// TIA Portal project "TAKT" (V15)

(* hardware
DEVICE "S7-1200 station_1"  S7-1200 Station
   slot 0: "Rack_0"  S7-1200 Rack  Rack  V1.0
   slot 1: "PLC_1"  CPU 1212C DC/DC/DC  6ES7 212-1AE40-0XB0  V4.2
*)

// ===== PLC "PLC_1"  CPU 1212C DC/DC/DC =====

VAR_GLOBAL   // PLC tag table "Default tag table"
   "PULSE1" AT %M0.0 : Bool;
   "PULSE_2" AT %M0.1 : Bool;
   "PULSE_4" AT %M0.2 : Bool;
   "PULSE3" AT %M0.3 : Bool;
END_VAR

TYPE "STOP_TIME"
   STRUCT
      BOTAO_ID : Int;
      DATE_INICIO : DTL;
      DATE_FIM : DTL;
   END_STRUCT;
END_TYPE

DATA_BLOCK "DIA_DA_SEMANA_DB"   // DB2
{ S7_Optimized_Access := 'TRUE' }
VERSION : 0.1
// stored: InstanceOfName DIA_DA_SEMANA
"DIA_DA_SEMANA"
BEGIN
END_DATA_BLOCK

DATA_BLOCK "Takt_Variavel_DB"   // DB4
{ S7_Optimized_Access := 'TRUE' }
VERSION : 0.1
// stored: InstanceOfName Takt_Variavel
"Takt_Variavel"
BEGIN
END_DATA_BLOCK

DATA_BLOCK "BANCO_DADOS_PARADAS"   // DB5
{ S7_Optimized_Access := 'TRUE' }
VERSION : 0.1
   VAR
      STOP_TIME : Array[0..1000] of "STOP_TIME";
   END_VAR
BEGIN
END_DATA_BLOCK

DATA_BLOCK "RELATORIO_DB"   // DB6
{ S7_Optimized_Access := 'TRUE' }
VERSION : 0.1
// stored: InstanceOfName RELATORIO
"RELATORIO"
BEGIN
END_DATA_BLOCK

DATA_BLOCK "TONR_DB"   // DB8
{ S7_Optimized_Access := 'TRUE' }
VERSION : 0.1
// stored: InstanceOfName TONR
"TONR"
BEGIN
END_DATA_BLOCK

// folder: System blocks/Program resources

DATA_BLOCK "Counter_DIA"   // DB1
{ S7_Optimized_Access := 'TRUE' }
AUTHOR : Simatic
FAMILY : IEC
NAME : CNTR
VERSION : 1.0
// stored: InstanceOfName IEC_COUNTER
"IEC_COUNTER"
BEGIN
END_DATA_BLOCK

DATA_BLOCK "Timer_RESET_TAKT"   // DB3
{ S7_Optimized_Access := 'TRUE' }
AUTHOR : Simatic
FAMILY : IEC
NAME : IEC_TMR
VERSION : 1.0
// stored: InstanceOfName IEC_TIMER
"IEC_TIMER"
BEGIN
END_DATA_BLOCK

// folder: (top level)

FUNCTION_BLOCK "Takt_Variavel"   // FB1, SCL
{ S7_Optimized_Access := 'TRUE' }
VERSION : 0.1
   VAR_INPUT
      IHM_SEGUNDA : Bool;   // BOTAO DA IHM DO DIA SEGUNDA-FEIRA
      IHM_TERCA : Bool;   // BOTAO DA IHM DO DIA TERÇA-FEIRA
      IHM_QUARTA : Bool;   // BOTAO DA IHM DO DIA QUARTA-FEIRA
      IHM_QUINTA : Bool;   // BOTAO DA IHM DO DIA QUINTA-FEIRA
      IHM_SEXTA : Bool;   // BOTAO DA IHM DO DIA SEXTA-FEIRA
      IHM_SABADO : Bool;   // BOTAO DA IHM DO DIA SABADO
      IHM_DOMINGO : Bool;   // BOTAO DA IHM DO DIA DOMINGO
      IHM_VALOR_TAKT : Int;   // VALOR DO TAKT NUMERO 1
      IHM_VALOR_TAKT_1 : Int;   // VALOR DO TAKT NUMERO 2
      IHM_VALOR_OBJETIVO : Int;   // VALOR DO OBJETIVO DO DIA SETADO NA IHM
      IHM_ALMOCO : Time_Of_Day;   // INICIO DO HORARIO DE ALMOÇO
      IHM_ALMOCO_FIM : Time_Of_Day;   // FIM DO HORARIO DE ALMOÇO
      IHM_JANTA : Time_Of_Day;   // INICIO DO HORARIO DE JANTA
      IHM_JANTA_FIM : Time_Of_Day;   // FIM DO HORARIO DE JANTA
      IHM_CAFE : Time_Of_Day;   // INICIO DO HORARIO DE CAFE
      IHM_CAFE_FIM : Time_Of_Day;   // FIM DO HORARIO DE CAFE
      IHM_INICIO_1TURNO : Time_Of_Day;   // INICIO DO 1 TURNO
      IHM_FIM_1TURNO : Time_Of_Day;   // FIM DO PRIMEIRO TURNO
      IHM_INICIO_2TURNO : Time_Of_Day;   // INICIO DO 2 TURNO
      IHM_FIM_2TURNO : Time_Of_Day;   // FIM DO 2 TURNO
      IHM_INICIO_3TURNO : Time_Of_Day;   // INICIO DO 3 TURNO
      IHM_FIM_3TURNO : Time_Of_Day;   // FIM DO 3 TURNO
      IHM_INICIO_PARADA : Time_Of_Day;   // INICIO DA PARADA RPOGRAMA
      IHM_FIM_PARADA : Time_Of_Day;   // FIM DA PARADA RPOGRAMA
      IHM_QUAL_TAKT : Int;   // QUAL O TAKT ESCOLHIDO
      ANDON_1 : Bool;   // BOTAO DE ANDON
      ANDON_2 : Bool;   // BOTAO DE ANDON
      ANDON_3 : Bool;   // BOTAO DE ANDON
      ANDON_4 : Bool;   // BOTAO DE ANDON
      ANDON_5 : Bool;   // BOTAO DE ANDON
      ANDON_6 : Bool;   // BOTAO DE ANDON
      ANDON_7 : Bool;   // BOTAO DE ANDON
      ANDON_8 : Bool;   // BOTAO DE ANDON
      ANDON_9 : Bool;   // BOTAO DE ANDON
      EMERGENCIA_1 : Bool;   // BOTAO DE EMERGENCIA OU STATUS DE EMERGENCIA
      EMERGENCIA_2 : Bool;   // BOTAO DE EMERGENCIA OU STATUS DE EMERGENCIA
      EMERGENCIA_3 : Bool;   // BOTAO DE EMERGENCIA OU STATUS DE EMERGENCIA
      EMERGENCIA_4 : Bool;   // BOTAO DE EMERGENCIA OU STATUS DE EMERGENCIA
      EMERGENCIA_5 : Bool;   // BOTAO DE EMERGENCIA OU STATUS DE EMERGENCIA
      EMERGENCIA_6 : Bool;   // BOTAO DE EMERGENCIA OU STATUS DE EMERGENCIA
      EMERGENCIA_7 : Bool;   // BOTAO DE EMERGENCIA OU STATUS DE EMERGENCIA
      EMERGENCIA_8 : Bool;   // BOTAO DE EMERGENCIA OU STATUS DE EMERGENCIA
      EMERGENCIA_9 : Bool;   // BOTAO DE EMERGENCIA OU STATUS DE EMERGENCIA
   END_VAR
   VAR_OUTPUT
      OUT_VALOR_TAKT : Int;   // VALOR DO TAKT EM INT
      OUT_VALOR_STOP_TIME : Int;   // VALOR TOTAL DO STOP TIME EM INT
      OUT_OBJETIVO : Int;   // VALOR DO OBJETIVO EM INT
      OUT_PRODUCAO_ATUAL : Int;   // VALOR DA PRODUCAO TOTAL EM INT
      OUT_DIA_DA_SEMANA : Int;   // DIA DA SEMANA EM INT DE 0 A 6
      OUT_DIA_DA_SEMANA_STRING : String;   // DIA DA SEMANA NO FORMATO DE STRING
      OUT_PARADA_PROGRAMADA : Bool;   // TEM PARADA PROGRAMADA
      OUT_REFEICAO : Bool;   // PARADA POR REFEIÇÃO
      OUT_EM_TURNO : Bool;   // EM TURNO
      OUT_SIRENE : Bool;   // TOCA SIRENE
   END_VAR
   VAR RETAIN
      Counter_PRODUCAO_ATUAL : CTU_INT;   // CONTADOR DE PRODUÇÃO
   END_VAR
   VAR
      Timer_RESET_STOP_TIME : TP_TIME;   // TIMER QUE RESETA O STOP TIME
      Timer_TAKT : TONR_TIME;   // TIMER DO TAKT
      Timer_STOP_TIME : TONR_TIME;   // TIMER DO STOP TIME
      S_ANDON : Array[1..8] of Bool;   // ARRAY DOS ANDONS
      S_EMERGENCIA : Array[1..8] of Bool;   // ARRAY DOS EMERGENCIAS
      S_VALOR_TAKT : Array[0..1] of Time;   // ARRAY DOS VALORES DE TAKT
      S_OBJETIVO_TURNO : Array[1..3] of Int;   // ARRAY DOS OBJETIVOS DOS TURNO
      TURNOS : Struct   // TURNOS
         S_INICIO_1TURNO : Time_Of_Day;
         S_FIM_1TURNO : Time_Of_Day;
         S_INICIO_2TURNO : Time_Of_Day;
         S_FIM_2TURNO : Time_Of_Day;
         S_INICIO_3TURNO : Time_Of_Day;
         S_FIM_3TURNO : Time_Of_Day;
         S_EM_TURNO : Bool;
      END_STRUCT;
      PARADAS : Struct   // PARADAS
         REFEIÇÃO : Bool;
         PROGRAMADA : Bool;
      END_STRUCT;
      PARADAS_REFEICOES : Struct   // PARADAS PARA REFEIÇÕES
         ALMOCO : Time_Of_Day;
         JANTA : Time_Of_Day;
         CAFE : Time_Of_Day;
         ALMOCO_FIM : Time_Of_Day := TOD#00:00:00;
         JANTA_FIM : Time_Of_Day := TOD#00:00:00;
         CAFE_FIM : Time_Of_Day := TOD#00:00:00;
      END_STRUCT;
      S_PROBLEMA : Bool;   // MEMORIA QUE É SETADA QUANDO TEM ALGUM ANDON OU EMERGENCIA ACIONADO
      S_DIA_ATIVA_TAKT : Bool;   // MEMORIA QUE VERIFICA O DIA DO TURNO ESTA ATIVO
      S_HORA_ATUAL : Time_Of_Day;   // CONTEM A HORA ATUAL
      S_TAKT_ON : Bool;   // MEMORIA DO TAKT LIGADO PARA CONTAR
      S_STOP_TIME_ON : Bool;   // MEMORIA DO STOP TIME LIGADO PARA CONTAR
      S_VALOR_TAKT_TIMER : Time;   // VALOR DO TAKT EM TIME
      S_RESET_TAKT : Bool;   // MEMORIA QUE RESETA O TAKT
      S_RESET_STOP_TIME : Bool;   // MEMORIA QUE RESETA O STOP TIME
      S_SIRENE : Bool;   // MEMORIA DA SIRENE E QUE SOMA A CONTA DO TOTAL PRODUZIDO
      S_VALOR_TAKT_ATUAL : Time;   // VALOR DO TAKT ATUAL EM TIME
      S_VALOR_STOP_TIME_ATUAL : Time;   // VALOR DO STOP TIME ATUAL EM TIME
      DIA_DA_SEMANA_STRING : String;
      DIA_DA_SEMANA_INT : Int;
      S_PRODUCAO_ATUAL : Int;   // MEMORIA PRODUÇÃO ATUAL
      S_PRODUCAO_FINALIZADA : Bool;   // PRODUÇÃO FINALIZADA
      S_CONVERT_TAKT : Int;   // MEMORIA QUE CONVERTE TIME PARA INT
      S_CONVERT_STOP_TIME : Int;   // MEMORIA QUE CONVERTE TIME PARA INT
   END_VAR
BEGIN
   (*
       ESTE BLOCO TEM POR FUNÇÃO CRIAR UM TAKT VARIAVEL DE FORMA QUE VOCÊ POSSA ESCOLHER MAIS DE UM VALOR DE TAKT 
   *)

   //JOGA AS ENTRADAS EM MEMORIAS LOCAIS 
   //--------ANDON--------//
   #S_ANDON[1] := #ANDON_1;
   #S_ANDON[2] := #ANDON_2;
   #S_ANDON[3] := #ANDON_3;
   #S_ANDON[4] := #ANDON_4;
   #S_ANDON[5] := #ANDON_5;
   #S_ANDON[6] := #ANDON_6;
   #S_ANDON[7] := #ANDON_7;
   #S_ANDON[8] := #ANDON_8;
   //--------TURNOS--------//
   #TURNOS.S_INICIO_1TURNO := #IHM_INICIO_1TURNO;
   #TURNOS.S_FIM_1TURNO := #IHM_FIM_1TURNO;
   #TURNOS.S_INICIO_2TURNO := #IHM_INICIO_2TURNO;
   #TURNOS.S_FIM_2TURNO := #IHM_FIM_2TURNO;
   #TURNOS.S_INICIO_3TURNO := #IHM_INICIO_3TURNO;
   #TURNOS.S_FIM_3TURNO := #IHM_FIM_3TURNO;
   //---------PARADA REFEIÇÃO---------//
   #PARADAS_REFEICOES.ALMOCO := #IHM_ALMOCO;
   #PARADAS_REFEICOES.ALMOCO_FIM := #IHM_ALMOCO_FIM;
   #PARADAS_REFEICOES.JANTA := #IHM_JANTA;
   #PARADAS_REFEICOES.JANTA_FIM := #IHM_JANTA_FIM;
   #PARADAS_REFEICOES.CAFE := #IHM_CAFE;
   #PARADAS_REFEICOES.CAFE_FIM := #IHM_CAFE_FIM;


   //-------------------------------------LOGICA PRINCIPAL DO BLOCO-------------------------------------//



   //TIMER DO TAKT 
   #Timer_TAKT(IN:=#S_TAKT_ON,
               R:= #S_RESET_TAKT,
               PT:=#S_VALOR_TAKT_TIMER,
               Q=>#S_SIRENE,
               ET=>#S_VALOR_TAKT_ATUAL);
   //TIMER DO STOP TIME
   #Timer_STOP_TIME(IN:=#S_STOP_TIME_ON,
                    R:=#S_RESET_STOP_TIME,
                    PT:=T#280000S,
                    ET=>#S_VALOR_STOP_TIME_ATUAL);
   // RESET TAKT

   "Timer_RESET_TAKT".TP(IN := (#TURNOS.S_EM_TURNO AND #S_DIA_ATIVA_TAKT AND NOT #PARADAS.PROGRAMADA
                         AND NOT #PARADAS.REFEIÇÃO AND NOT #S_PROBLEMA AND #Timer_TAKT.ET = #S_VALOR_TAKT_TIMER)
                         OR(#TURNOS.S_INICIO_1TURNO = #S_HORA_ATUAL)
                         OR (#TURNOS.S_INICIO_2TURNO = #S_HORA_ATUAL)
                         OR (#TURNOS.S_INICIO_3TURNO = #S_HORA_ATUAL),
                         PT := T#100MS,
                         Q => #S_RESET_TAKT);

   // RESET STOP TIME    
   #Timer_RESET_STOP_TIME(IN := (#TURNOS.S_FIM_1TURNO = #S_HORA_ATUAL) OR
                          (#TURNOS.S_FIM_2TURNO = #S_HORA_ATUAL) OR
                          (#TURNOS.S_FIM_3TURNO = #S_HORA_ATUAL),
                          PT := T#100MS,
                          Q => #S_RESET_STOP_TIME);
   //CONTADOR DE PRODUÇÃO ATUAL
   #Counter_PRODUCAO_ATUAL(CU := #S_SIRENE,
                           R := (#TURNOS.S_INICIO_1TURNO = #S_HORA_ATUAL)
                           OR (#TURNOS.S_INICIO_2TURNO = #S_HORA_ATUAL)
                           OR (#TURNOS.S_INICIO_3TURNO = #S_HORA_ATUAL),
                           PV := #IHM_VALOR_OBJETIVO,
                           Q => #S_PRODUCAO_FINALIZADA,
                           CV => #S_PRODUCAO_ATUAL);


   //INFORMA O DIA DA SEMANA COMO INTEIRO E STRING 0 Á 6 / SEGUNDA Á DOMINGO
   "DIA_DA_SEMANA_DB"(OUT_DIA_DA_SEMANA_STRING=>#DIA_DA_SEMANA_STRING,
                      OUT_DIA_DA_SEMANA_INT=>#DIA_DA_SEMANA_INT,
                      OUT_HORA_ATUAL=>#S_HORA_ATUAL);



   //VERIFICA AS BOTOEIRAS DE ANDON E OS EMERGENCIAS 
   IF (#S_ANDON[1] OR #S_ANDON[2] OR #S_ANDON[3] OR #S_ANDON[4] OR #S_ANDON[5] OR #S_ANDON[6] OR #S_ANDON[7] OR #S_ANDON[8]) OR
       (#S_EMERGENCIA[1] OR #S_EMERGENCIA[2] OR #S_EMERGENCIA[3] OR #S_EMERGENCIA[4] OR #S_EMERGENCIA[5] OR #S_EMERGENCIA[6] OR #S_EMERGENCIA[7] OR #S_EMERGENCIA[8]) THEN
       #S_PROBLEMA := 1;
   ELSE
       #S_PROBLEMA := 0;
   END_IF;

   //VERIFICA SE O DIA DA SEMANA ESTA ATIVO PARA RODAR O TAKT 
   IF #IHM_SEGUNDA AND (#DIA_DA_SEMANA_INT = 0) THEN

       #S_DIA_ATIVA_TAKT := 1;

   ELSIF(#IHM_TERCA AND (#DIA_DA_SEMANA_INT = 1)) THEN

       #S_DIA_ATIVA_TAKT := 1;

   ELSIF(#IHM_QUARTA AND (#DIA_DA_SEMANA_INT = 2)) THEN

       #S_DIA_ATIVA_TAKT := 1;

   ELSIF(#IHM_QUINTA AND (#DIA_DA_SEMANA_INT = 3) )THEN

       #S_DIA_ATIVA_TAKT := 1;

   ELSIF(#IHM_SEXTA AND (#DIA_DA_SEMANA_INT = 4) )THEN

       #S_DIA_ATIVA_TAKT := 1;

   ELSIF(#IHM_SABADO AND (#DIA_DA_SEMANA_INT = 5) )THEN

       #S_DIA_ATIVA_TAKT := 1;

   ELSIF(#IHM_DOMINGO AND (#DIA_DA_SEMANA_INT = 6)) THEN

       #S_DIA_ATIVA_TAKT := 1;

   ELSE

       #S_DIA_ATIVA_TAKT := 0;

   END_IF;


   //VERIFICA O HORARIO DE PARADA (ALMOÇO,JANTA,CAFÉ E MUDANÇAS DE TURNO)

   IF #S_HORA_ATUAL >= #PARADAS_REFEICOES.ALMOCO AND #S_HORA_ATUAL <= #PARADAS_REFEICOES.ALMOCO_FIM  THEN
       #PARADAS.REFEIÇÃO := 1;
       ;
   ELSIF #S_HORA_ATUAL >= #PARADAS_REFEICOES.JANTA AND #S_HORA_ATUAL <= #PARADAS_REFEICOES.JANTA_FIM  THEN
       #PARADAS.REFEIÇÃO := 1;
       ;
   ELSIF #S_HORA_ATUAL >= #PARADAS_REFEICOES.CAFE AND #S_HORA_ATUAL <= #PARADAS_REFEICOES.CAFE_FIM  THEN
       #PARADAS.REFEIÇÃO := 1;
       ;
   ELSE
       #PARADAS.REFEIÇÃO := 0;
   END_IF;

   // VERIFICA PARADAS PROGRAMADAS(SINDICATO, GINASTICA ELABORAL E ETC...)
   IF #S_HORA_ATUAL >= #IHM_INICIO_PARADA AND #S_HORA_ATUAL <= #IHM_FIM_PARADA THEN
       #PARADAS.PROGRAMADA := 1;
   ELSE
       #PARADAS.PROGRAMADA := 0;
   END_IF;


   // VERIFICA HORARIO DE PRODUÇÃO
   IF #S_HORA_ATUAL >= #TURNOS.S_INICIO_1TURNO AND #S_HORA_ATUAL <= #TURNOS.S_FIM_1TURNO THEN
       #TURNOS.S_EM_TURNO := 1;

   ELSIF  #S_HORA_ATUAL >= #TURNOS.S_INICIO_2TURNO AND #S_HORA_ATUAL <= #TURNOS.S_FIM_2TURNO THEN
       #TURNOS.S_EM_TURNO := 1;

   ELSIF  #S_HORA_ATUAL >= #TURNOS.S_INICIO_3TURNO AND #S_HORA_ATUAL <= #TURNOS.S_FIM_3TURNO THEN
       #TURNOS.S_EM_TURNO := 1;

   ELSE
       #TURNOS.S_EM_TURNO := 0;
       ;
   END_IF;


   // VERIFICA SE ESTÁ TUDO OK PARA CONTAR O TAKT

   IF #TURNOS.S_EM_TURNO AND #S_DIA_ATIVA_TAKT AND NOT #PARADAS.PROGRAMADA AND NOT #PARADAS.REFEIÇÃO AND #Timer_TAKT.ET < #S_VALOR_TAKT_TIMER AND NOT #S_PRODUCAO_FINALIZADA THEN
       #S_TAKT_ON := 1;
       #S_STOP_TIME_ON := 0;
   ELSIF #TURNOS.S_EM_TURNO AND #S_DIA_ATIVA_TAKT AND NOT #PARADAS.PROGRAMADA AND NOT #PARADAS.REFEIÇÃO AND #S_PROBLEMA AND #Timer_TAKT.ET = #S_VALOR_TAKT_TIMER THEN
       #S_TAKT_ON := 0;
       #S_STOP_TIME_ON := 1;
   ELSE
       #S_TAKT_ON := 0;
       #S_STOP_TIME_ON := 0;
   END_IF;


   // ESCOLHE QUAL O VALOR DE TAKT SE É O 1 OU O N

   CASE #IHM_QUAL_TAKT OF
       1:
           #S_VALOR_TAKT[0] := INT_TO_TIME(#IHM_VALOR_TAKT) * 1000;
           #S_VALOR_TAKT_TIMER := #S_VALOR_TAKT[0]; ;
       2:
           #S_VALOR_TAKT[1] := INT_TO_TIME(#IHM_VALOR_TAKT_1) * 1000;
           #S_VALOR_TAKT_TIMER  := #S_VALOR_TAKT[1];
       ELSE  
           #S_VALOR_TAKT_TIMER  := t#0S;
   END_CASE;

   //CONVERTE O TAKT DE TIME PARA INT
   #S_CONVERT_TAKT := TIME_TO_INT(#S_VALOR_TAKT_ATUAL)/1000;
   //CONVERTE O STOP TIME DE TIME PARA INT
   #S_CONVERT_STOP_TIME:= TIME_TO_INT(#S_VALOR_STOP_TIME_ATUAL)/1000;

   //JOGA AS MEMORIAS LOCAIS NAS SAIDAS

   #OUT_VALOR_TAKT := #S_CONVERT_TAKT;
   #OUT_VALOR_TAKT:= #IHM_VALOR_TAKT - #OUT_VALOR_TAKT;
   #OUT_VALOR_STOP_TIME := #S_CONVERT_STOP_TIME;
   #OUT_OBJETIVO := #IHM_VALOR_OBJETIVO;
   #OUT_PRODUCAO_ATUAL := #S_PRODUCAO_ATUAL;
   #OUT_DIA_DA_SEMANA := #DIA_DA_SEMANA_INT;
   #OUT_DIA_DA_SEMANA_STRING := #DIA_DA_SEMANA_STRING;
   #OUT_PARADA_PROGRAMADA := #PARADAS.PROGRAMADA;
   #OUT_REFEICAO := #PARADAS.REFEIÇÃO;
   #OUT_EM_TURNO := #TURNOS.S_EM_TURNO;
   #OUT_SIRENE := #S_SIRENE;
END_FUNCTION_BLOCK

FUNCTION_BLOCK "DIA_DA_SEMANA"   // FB2, SCL
{ S7_Optimized_Access := 'TRUE' }
VERSION : 0.1
   VAR_OUTPUT
      OUT_DIA_DA_SEMANA_STRING : String;
      OUT_DIA_DA_SEMANA_INT : Int;
      OUT_HORA_ATUAL : Time_Of_Day;
   END_VAR
   VAR
      S_ERRO_DE_LEITURA_DATA : Int;
      S_MEIA_NOITE : Time_Of_Day := TOD#23:59:00;
      S_MEIA_NOITE_1 : Time_Of_Day := TOD#00:01:00;
      S_HORARIO_ATUAL : Time_Of_Day;
      S_DATA_DO_DIA : DTL;
      S_ATIVA_CONTAR : Bool;
      S_CONTAGEM : Int;
      S_DIA_DA_SEMANA : String;
      S_RESET_CONTADOR : Bool;
   END_VAR
BEGIN


   //FAZ A LEITURA DA DATA DO SISTEMA 
   #S_ERRO_DE_LEITURA_DATA := RD_SYS_T(#S_DATA_DO_DIA);
   // TRANSFORMA PARA A VARIAVEL TIMEOFDAY
   #S_HORARIO_ATUAL := DTL_TO_TOD(#S_DATA_DO_DIA);




   // CONTADOR AUXILIAR PARA SABER O DIA
   "Counter_DIA".CTU(CU := #S_ATIVA_CONTAR,
                     R:=#S_RESET_CONTADOR,
                     PV := 6,
                     CV=>#S_CONTAGEM);
   // ROTINA PARA SABER O DIA DA SEMANA 
   IF (#S_HORARIO_ATUAL >= #S_MEIA_NOITE AND #S_HORARIO_ATUAL <= #S_MEIA_NOITE_1) THEN
       #S_ATIVA_CONTAR := 1;
   ELSE
       #S_ATIVA_CONTAR := 0;
       ;
   END_IF;
   // CONFERE A DATA E RESETA O CONTADOR
   IF #S_CONTAGEM = 6 AND (#S_HORARIO_ATUAL >= #S_MEIA_NOITE AND #S_HORARIO_ATUAL <= #S_MEIA_NOITE_1) THEN
       #S_RESET_CONTADOR := 1;
   ELSE
       #S_RESET_CONTADOR := 0;
       ;
   END_IF;

   //DÁ NOME AOS DIAS
   CASE #S_CONTAGEM OF
       0:  //SEGUNTA-FEIRA
           #S_DIA_DA_SEMANA := 'SEGUNDA-FEIRA';
       1:  //TERÇA-FEIRA
           #S_DIA_DA_SEMANA := 'TERCA-FEIRA';
           ;
       2:  //QUARTA-FEIRA
           #S_DIA_DA_SEMANA := 'QUARTA-FEIRA';
           ;
       3:  //QUINTA-FEIRA
           #S_DIA_DA_SEMANA := 'QUINTA-FEIRA';
           ;
       4:  //SEXTA-FEIRA
           #S_DIA_DA_SEMANA := 'SEXTA-FEIRA';
           ;
       5:  //SABADO
           #S_DIA_DA_SEMANA := 'SABADO';
           ;
       6:  //DOMINGO
           #S_DIA_DA_SEMANA := 'DOMINGO';
           ;
       ELSE  // Statement section ELSE
           #S_DIA_DA_SEMANA := 'NONE';
   END_CASE;


   // JOGA AS MEMORIAS NAS SAIDA

   #OUT_DIA_DA_SEMANA_STRING := #S_DIA_DA_SEMANA;
   #OUT_DIA_DA_SEMANA_INT := #S_CONTAGEM;
   #OUT_HORA_ATUAL := #S_HORARIO_ATUAL;
END_FUNCTION_BLOCK

FUNCTION_BLOCK "DIAGNOSE"   // FB3, SCL
{ S7_Optimized_Access := 'TRUE' }
VERSION : 0.1
BEGIN
END_FUNCTION_BLOCK

FUNCTION_BLOCK "RELATORIO"   // FB4, SCL
{ S7_Optimized_Access := 'TRUE' }
VERSION : 0.1
   VAR_INPUT
      ANDON_1 : Bool;
      ANDON_2 : Bool;
      ANDON_3 : Bool;
      ANDON_4 : Bool;
      ANDON_5 : Bool;
      ANDON_6 : Bool;
      ANDON_7 : Bool;
      ANDON_8 : Bool;
      ANDON_9 : Bool;
      EMERGENCIA_1 : Bool;
      EMERGENCIA_2 : Bool;
      EMERGENCIA_3 : Bool;
      EMERGENCIA_4 : Bool;
      EMERGENCIA_5 : Bool;
      EMERGENCIA_6 : Bool;
      EMERGENCIA_7 : Bool;
      EMERGENCIA_8 : Bool;
      EMERGENCIA_9 : Bool;
      ANDON_10 : Bool;
      ANDON_11 : Bool;
      ANDON_12 : Bool;
      ANDON_13 : Bool;
      ANDON_14 : Bool;
      ANDON_15 : Bool;
      ANDON_16 : Bool;
      ANDON_17 : Bool;
      ANDON_18 : Bool;
      EMERGENCIA_10 : Bool;
      EMERGENCIA_11 : Bool;
      EMERGENCIA_12 : Bool;
      EMERGENCIA_13 : Bool;
      EMERGENCIA_14 : Bool;
      EMERGENCIA_15 : Bool;
      EMERGENCIA_16 : Bool;
      EMERGENCIA_17 : Bool;
      EMERGENCIA_18 : Bool;
   END_VAR
   VAR
      N : Int := 0;
      HORA_ATUAL : DTL;
      ERRO_DTL : Int;
   END_VAR
BEGIN

   #ERRO_DTL := RD_SYS_T(#HORA_ATUAL);

   IF #ANDON_1 THEN

       "BANCO_DADOS_PARADAS".STOP_TIME[#N].BOTAO_ID := 1;
       "BANCO_DADOS_PARADAS".STOP_TIME[#N].DATE_INICIO := #HORA_ATUAL;

        #N := #N+1;
        ;
    ELSIF #ANDON_2 THEN

        "BANCO_DADOS_PARADAS".STOP_TIME[#N].BOTAO_ID := 2;
        "BANCO_DADOS_PARADAS".STOP_TIME[#N].DATE_INICIO := #HORA_ATUAL;

        #N := #N + 1;
    ELSIF #ANDON_3 THEN

        "BANCO_DADOS_PARADAS".STOP_TIME[#N].BOTAO_ID := 3;
        "BANCO_DADOS_PARADAS".STOP_TIME[#N].DATE_INICIO := #HORA_ATUAL;

        #N := #N + 1;
    ELSIF #ANDON_4 THEN

        "BANCO_DADOS_PARADAS".STOP_TIME[#N].BOTAO_ID := 4;
        "BANCO_DADOS_PARADAS".STOP_TIME[#N].DATE_INICIO := #HORA_ATUAL;

        #N := #N + 1;
    ELSIF #ANDON_5 THEN

        "BANCO_DADOS_PARADAS".STOP_TIME[#N].BOTAO_ID := 5;
        "BANCO_DADOS_PARADAS".STOP_TIME[#N].DATE_INICIO := #HORA_ATUAL;

        #N := #N + 1;
    ELSIF #ANDON_6 THEN

        "BANCO_DADOS_PARADAS".STOP_TIME[#N].BOTAO_ID := 6;
        "BANCO_DADOS_PARADAS".STOP_TIME[#N].DATE_INICIO := #HORA_ATUAL;

        #N := #N + 1;
    ELSIF #ANDON_7 THEN

        "BANCO_DADOS_PARADAS".STOP_TIME[#N].BOTAO_ID := 7;
        "BANCO_DADOS_PARADAS".STOP_TIME[#N].DATE_INICIO := #HORA_ATUAL;

        #N := #N + 1;
    ELSIF #ANDON_8 THEN

        "BANCO_DADOS_PARADAS".STOP_TIME[#N].BOTAO_ID := 8;
        "BANCO_DADOS_PARADAS".STOP_TIME[#N].DATE_INICIO := #HORA_ATUAL;

        #N := #N + 1;
    ELSIF #ANDON_9 THEN

        "BANCO_DADOS_PARADAS".STOP_TIME[#N].BOTAO_ID := 9;
        "BANCO_DADOS_PARADAS".STOP_TIME[#N].DATE_INICIO := #HORA_ATUAL;

        #N := #N + 1;
    ELSIF #EMERGENCIA_1 THEN

        "BANCO_DADOS_PARADAS".STOP_TIME[#N].BOTAO_ID := 10;
        "BANCO_DADOS_PARADAS".STOP_TIME[#N].DATE_INICIO := #HORA_ATUAL;

        #N := #N + 1;
    ELSIF #EMERGENCIA_2 THEN

        "BANCO_DADOS_PARADAS".STOP_TIME[#N].BOTAO_ID := 11;
        "BANCO_DADOS_PARADAS".STOP_TIME[#N].DATE_INICIO := #HORA_ATUAL;

        #N := #N + 1;
    ELSIF #EMERGENCIA_3 THEN

        "BANCO_DADOS_PARADAS".STOP_TIME[#N].BOTAO_ID := 12;
        "BANCO_DADOS_PARADAS".STOP_TIME[#N].DATE_INICIO := #HORA_ATUAL;

        #N := #N + 1;
    ELSIF #EMERGENCIA_4 THEN

        "BANCO_DADOS_PARADAS".STOP_TIME[#N].BOTAO_ID := 13;
        "BANCO_DADOS_PARADAS".STOP_TIME[#N].DATE_INICIO := #HORA_ATUAL;

        #N := #N + 1;
    ELSIF #EMERGENCIA_5 THEN

        "BANCO_DADOS_PARADAS".STOP_TIME[#N].BOTAO_ID := 14;
        "BANCO_DADOS_PARADAS".STOP_TIME[#N].DATE_INICIO := #HORA_ATUAL;

        #N := #N + 1;
    ELSIF #EMERGENCIA_6 THEN

        "BANCO_DADOS_PARADAS".STOP_TIME[#N].BOTAO_ID := 15;
        "BANCO_DADOS_PARADAS".STOP_TIME[#N].DATE_INICIO := #HORA_ATUAL;

        #N := #N + 1;
    ELSIF #EMERGENCIA_7 THEN

        "BANCO_DADOS_PARADAS".STOP_TIME[#N].BOTAO_ID := 16;
        "BANCO_DADOS_PARADAS".STOP_TIME[#N].DATE_INICIO := #HORA_ATUAL;

        #N := #N + 1;
    ELSIF #EMERGENCIA_8 THEN

        "BANCO_DADOS_PARADAS".STOP_TIME[#N].BOTAO_ID := 17;
        "BANCO_DADOS_PARADAS".STOP_TIME[#N].DATE_INICIO := #HORA_ATUAL;

        #N := #N + 1;
    ELSIF #EMERGENCIA_9 THEN

        "BANCO_DADOS_PARADAS".STOP_TIME[#N].BOTAO_ID := 18;
        "BANCO_DADOS_PARADAS".STOP_TIME[#N].DATE_INICIO := #HORA_ATUAL;

        #N := #N + 1;
    ELSE
        ;

   END_IF;
   IF #N = 1000 THEN
       #N := 0;
       ;
   END_IF;
END_FUNCTION_BLOCK

FUNCTION_BLOCK "TONR"   // FB5, SCL
{ S7_Optimized_Access := 'TRUE' }
VERSION : 0.1
   VAR_INPUT
      IN : Bool;
      R : Bool;
      PT : Time;
   END_VAR
   VAR_OUTPUT
      ET : Time;
      Q : Bool;
   END_VAR
   VAR
      "Timer" : TON_TIME;
   END_VAR
   VAR RETAIN
      S_Timer : Time;
   END_VAR
   VAR
      S_PT : Time;
      R_TRIG_Instance : R_TRIG;
      S_ET : Time;
   END_VAR
BEGIN
   #R_TRIG_Instance(CLK := #IN);
   IF #PT > #S_Timer AND #S_Timer > T#0s AND #R_TRIG_Instance.Q THEN
       #S_PT := #PT - #S_Timer;
   ELSIF #Timer.Q THEN
       #S_PT := #PT;
       #S_Timer := T#0s;
   END_IF;





   #Timer(IN:=#IN,
          PT:= #S_PT,
          Q=>#Q,
          ET=>#S_ET);


   IF #S_ET <= #PT AND #IN THEN
       #S_Timer := #S_ET ;
   ELSIF #Timer.Q THEN
       #S_Timer := T#0s;
       #S_PT := #PT;
   END_IF;

   #ET := #S_PT;
END_FUNCTION_BLOCK

ORGANIZATION_BLOCK "Main"   // OB1, LAD, ProgramCycle
TITLE = "Main Program Sweep (Cycle)"
{ S7_Optimized_Access := 'TRUE' }
VERSION : 0.1
   VAR_INPUT
      Initial_Call : Bool;   // Initial call of this OB
      Remanence : Bool;   // =True, if remanent data are available
   END_VAR
   VAR_TEMP   // added for the SCL form of the ladder/FBD networks
      _w1 : Bool;
      _w2 : Bool;
   END_VAR
BEGIN

REGION Network 1
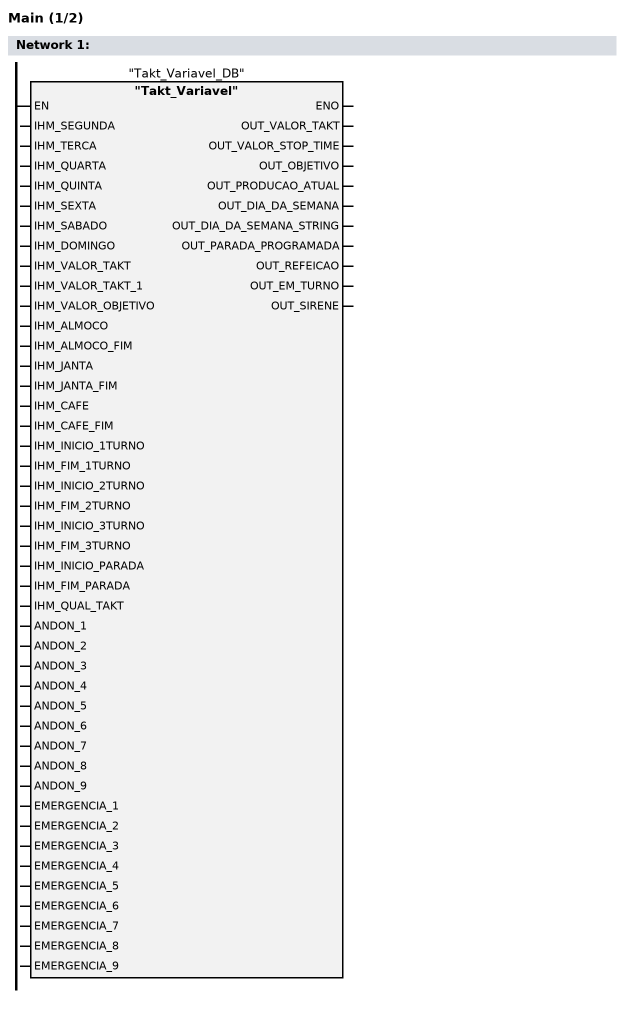
   RUNG wire#powerrail
      "Takt_Variavel_DB"(IHM_SEGUNDA :=, IHM_TERCA :=, IHM_QUARTA :=, IHM_QUINTA :=, IHM_SEXTA :=, IHM_SABADO :=, IHM_DOMINGO :=, IHM_VALOR_TAKT :=, IHM_VALOR_TAKT_1 :=, IHM_VALOR_OBJETIVO :=, IHM_ALMOCO :=, IHM_ALMOCO_FIM :=, IHM_JANTA :=, IHM_JANTA_FIM :=, IHM_CAFE :=, IHM_CAFE_FIM :=, IHM_INICIO_1TURNO :=, IHM_FIM_1TURNO :=, IHM_INICIO_2TURNO :=, IHM_FIM_2TURNO :=, IHM_INICIO_3TURNO :=, IHM_FIM_3TURNO :=, IHM_INICIO_PARADA :=, IHM_FIM_PARADA :=, IHM_QUAL_TAKT :=, ANDON_1 :=, ANDON_2 :=, ANDON_3 :=, ANDON_4 :=, ANDON_5 :=, ANDON_6 :=, ANDON_7 :=, ANDON_8 :=, ANDON_9 :=, EMERGENCIA_1 :=, EMERGENCIA_2 :=, EMERGENCIA_3 :=, EMERGENCIA_4 :=, EMERGENCIA_5 :=, EMERGENCIA_6 :=, EMERGENCIA_7 :=, EMERGENCIA_8 :=, EMERGENCIA_9 :=, OUT_VALOR_TAKT =>, OUT_VALOR_STOP_TIME =>, OUT_OBJETIVO =>, OUT_PRODUCAO_ATUAL =>, OUT_DIA_DA_SEMANA =>, OUT_DIA_DA_SEMANA_STRING =>, OUT_PARADA_PROGRAMADA =>, OUT_REFEICAO =>, OUT_EM_TURNO =>, OUT_SIRENE =>)
   END_RUNG
   // the same network as SCL:
   "Takt_Variavel_DB"();   // "Takt_Variavel"
END_REGION

REGION Network 2
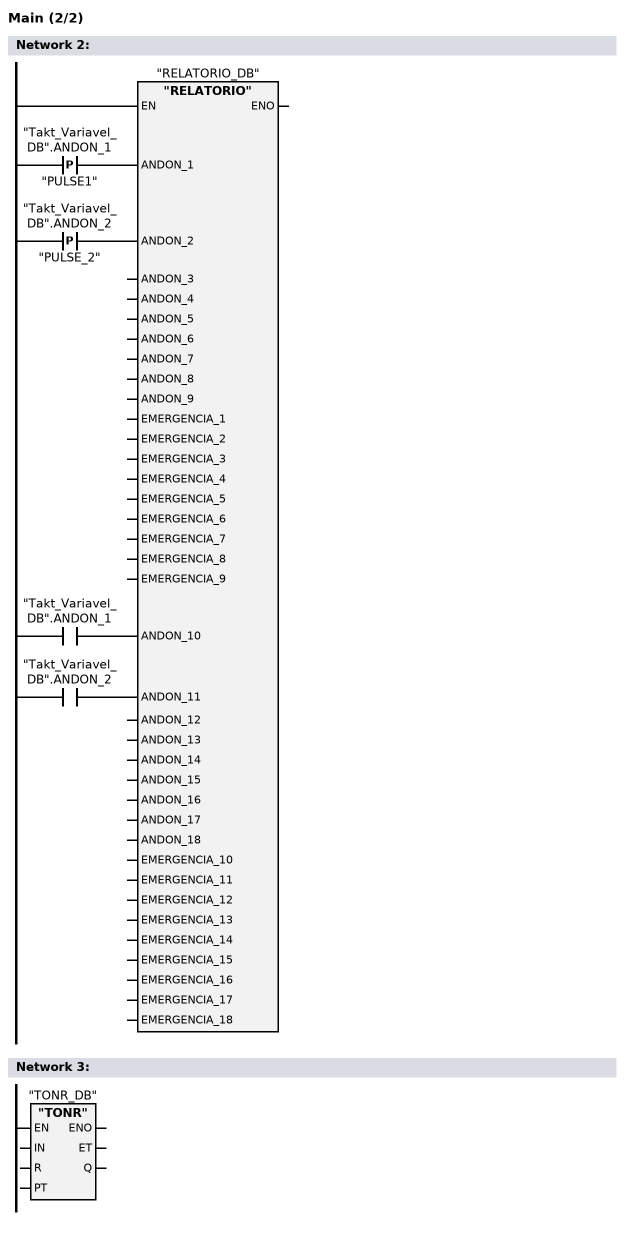
   RUNG wire#powerrail
      "RELATORIO_DB"(ANDON_1 := wire#w1, ANDON_2 := wire#w2, ANDON_10 := wire#w3, ANDON_11 := wire#w4, ANDON_3 :=, ANDON_4 :=, ANDON_5 :=, ANDON_6 :=, ANDON_7 :=, ANDON_8 :=, ANDON_9 :=, EMERGENCIA_1 :=, EMERGENCIA_2 :=, EMERGENCIA_3 :=, EMERGENCIA_4 :=, EMERGENCIA_5 :=, EMERGENCIA_6 :=, EMERGENCIA_7 :=, EMERGENCIA_8 :=, EMERGENCIA_9 :=, ANDON_12 :=, ANDON_13 :=, ANDON_14 :=, ANDON_15 :=, ANDON_16 :=, ANDON_17 :=, ANDON_18 :=, EMERGENCIA_10 :=, EMERGENCIA_11 :=, EMERGENCIA_12 :=, EMERGENCIA_13 :=, EMERGENCIA_14 :=, EMERGENCIA_15 :=, EMERGENCIA_16 :=, EMERGENCIA_17 :=, EMERGENCIA_18 :=)
   END_RUNG
   RUNG wire#powerrail
      P_Contact(operand := "Takt_Variavel_DB".ANDON_1, bit := "PULSE1")
   END_RUNG wire#w1
   RUNG wire#powerrail
      P_Contact(operand := "Takt_Variavel_DB".ANDON_2, bit := "PULSE_2")
   END_RUNG wire#w2
   RUNG wire#powerrail
      Contact( "Takt_Variavel_DB".ANDON_1 )
   END_RUNG wire#w3
   RUNG wire#powerrail
      Contact( "Takt_Variavel_DB".ANDON_2 )
   END_RUNG wire#w4
   // the same network as SCL:
   #_w1 := "Takt_Variavel_DB".ANDON_1 AND NOT "PULSE1";   // rising edge of "Takt_Variavel_DB".ANDON_1
   "PULSE1" := "Takt_Variavel_DB".ANDON_1;
   #_w2 := "Takt_Variavel_DB".ANDON_2 AND NOT "PULSE_2";   // rising edge of "Takt_Variavel_DB".ANDON_2
   "PULSE_2" := "Takt_Variavel_DB".ANDON_2;
   "RELATORIO_DB"(ANDON_1 := #_w1,   // "RELATORIO"
                  ANDON_2 := #_w2,
                  ANDON_10 := "Takt_Variavel_DB".ANDON_1,
                  ANDON_11 := "Takt_Variavel_DB".ANDON_2);
END_REGION

REGION Network 3
   RUNG wire#powerrail
      "TONR_DB"(IN :=, R :=, PT :=, ET =>, Q =>)
   END_RUNG
   // the same network as SCL:
   "TONR_DB"();   // "TONR"
END_REGION
END_ORGANIZATION_BLOCK